// TIA Portal project "Ejercicio3" (V15.1)

(* hardware
DEVICE "S7-1200 station_2"  S7-1200 Station
   slot 0: "Rack_0"  S7-1200 Rack  Rack  V1.0
   slot 1: "PLC_0"  CPU 1215C AC/DC/Rly  6ES7 215-1BG40-0XB0  V4.2
DEVICE "HMI_0"  KTP700 Basic PN
   slot 0: "HMI_0"  KTP700 Basic PN  6AV2 123-2GB03-0AX0  15.1.0.0
   slot 1: "HMI_RT_1"  KTP700 Basic PN  6AV2 123-2GB03-0AX0  15.1.0.0
   slot 5: "HMI_0.IE_CP_1"  PROFINET Interface  15.0.1.0
      slot 1: "Interfaz PROFINET_1"  PROFINET Interface
         slot 1: "Port_1"  Port
*)

// ===== PLC "PLC_0"  CPU 1215C AC/DC/Rly =====

VAR_GLOBAL   // PLC tag table "Tabla de variables estándar"
   "Marcha" AT %M0.0 : Bool;
   "Paro" AT %M0.1 : Bool;
   "Pila de pales en la entrada" AT %M0.2 : Bool;
   "Pila de pale en desapilador" AT %M0.3 : Bool;
   "Palé en rodillos de salida" AT %M0.4 : Bool;
   "Cilindro subir pilas pales reposo" AT %M0.5 : Bool;
   "Cilindro subir pilas pales arriba" AT %M0.6 : Bool;
   "Cilindro uña sujetar pila reposo" AT %M0.7 : Bool;
   "Cilindro uña sujetar pila extendida" AT %M1.0 : Bool;
   "Freno pila recogido" AT %M1.1 : Bool;
   "Freno pila extendido" AT %M1.2 : Bool;
   "Motor rodillos entrada pilas" AT %M10.0 : Bool;
   "Motor rodillos desapilador" AT %M10.1 : Bool;
   "Motor rodillos salida de palé" AT %M10.2 : Bool;
   "Cilindro subir pila" AT %M10.3 : Bool;
   "Cilindro uñas sujetar pila" AT %M10.4 : Bool;
   "Cilindro freno" AT %M10.5 : Bool;
   "Permiso de extraccion de palé" AT %M2.0 : Bool;
END_VAR

// folder: System blocks/Program resources

DATA_BLOCK "IEC_Timer_0_DB"   // DB1
{ S7_Optimized_Access := 'TRUE' }
AUTHOR : Simatic
FAMILY : IEC
NAME : IEC_TMR
VERSION : 1.0
// stored: InstanceOfName IEC_TIMER
"IEC_TIMER"
BEGIN
END_DATA_BLOCK

DATA_BLOCK "IEC_Timer_0_DB_1"   // DB2
{ S7_Optimized_Access := 'TRUE' }
AUTHOR : Simatic
FAMILY : IEC
NAME : IEC_TMR
VERSION : 1.0
// stored: InstanceOfName IEC_TIMER
"IEC_TIMER"
BEGIN
END_DATA_BLOCK

DATA_BLOCK "IEC_Timer_0_DB_2"   // DB3
{ S7_Optimized_Access := 'TRUE' }
AUTHOR : Simatic
FAMILY : IEC
NAME : IEC_TMR
VERSION : 1.0
// stored: InstanceOfName IEC_TIMER
"IEC_TIMER"
BEGIN
END_DATA_BLOCK

// folder: (top level)

ORGANIZATION_BLOCK "Main"   // OB1, LAD, ProgramCycle
TITLE = "Main Program Sweep (Cycle)"
{ S7_Optimized_Access := 'TRUE' }
VERSION : 0.1
   VAR_INPUT
      Initial_Call : Bool;   // Initial call of this OB
      Remanence : Bool;   // =True, if remanent data are available
   END_VAR
BEGIN

REGION Network 1
   // Tenemos  un  pulsador  de  marcha  uno  de  paro  para  el  sistema.  Si  se  pulsa  el  paro  la  secuencia  se detiene continuando en el mismo punto cuando se pulse marcha de nuevo.
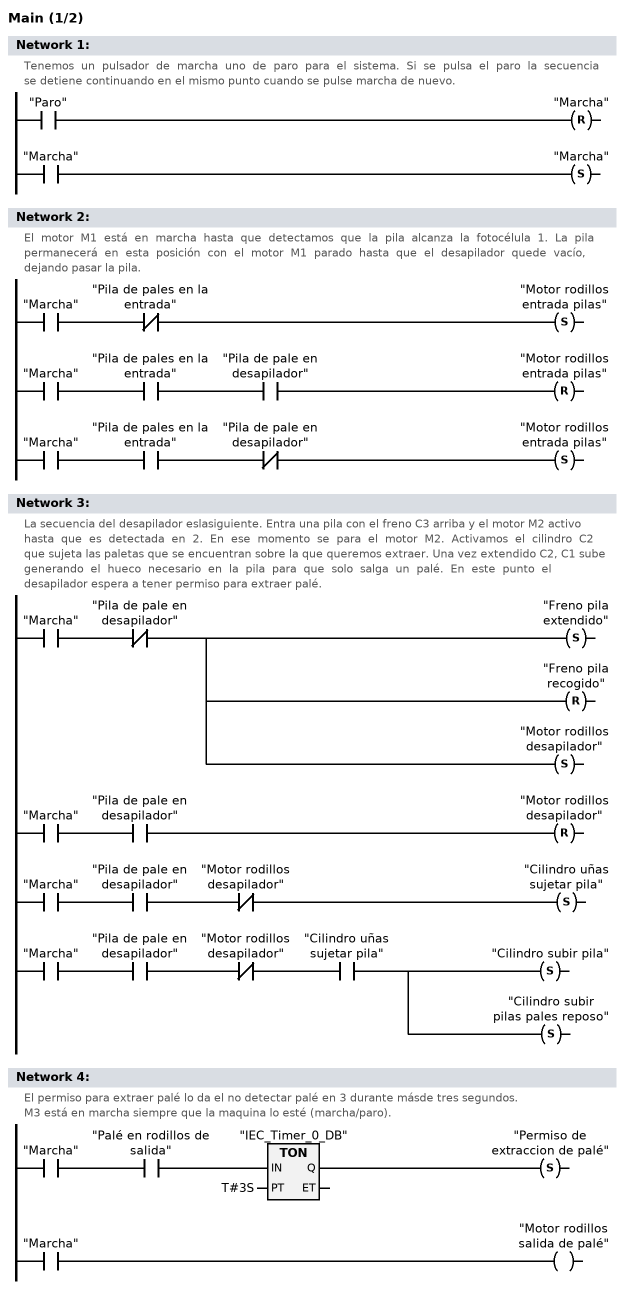
   RUNG wire#powerrail
      Contact( "Paro" )
      R_Coil( "Marcha" )
   END_RUNG
   RUNG wire#powerrail
      Contact( "Marcha" )
      S_Coil( "Marcha" )
   END_RUNG
   // the same network as SCL:
   IF "Paro" THEN "Marcha" := FALSE; END_IF;
   IF "Marcha" THEN "Marcha" := TRUE; END_IF;
END_REGION

REGION Network 2
   // El  motor  M1  está  en  marcha  hasta  que  detectamos  que  la  pila  alcanza  la  fotocélula  1.  La  pila permanecerá  en  esta  posición  con  el  motor  M1  parado  hasta  que  el  desapilador  quede  vacío, dejando pasar la pila.
   RUNG wire#powerrail
      Contact( "Marcha" )
      I_Contact( "Pila de pales en la entrada" )
      S_Coil( "Motor rodillos entrada pilas" )
   END_RUNG
   RUNG wire#powerrail
      Contact( "Marcha" )
      Contact( "Pila de pales en la entrada" )
      Contact( "Pila de pale en desapilador" )
      R_Coil( "Motor rodillos entrada pilas" )
   END_RUNG
   RUNG wire#powerrail
      Contact( "Marcha" )
      Contact( "Pila de pales en la entrada" )
      I_Contact( "Pila de pale en desapilador" )
      S_Coil( "Motor rodillos entrada pilas" )
   END_RUNG
   // the same network as SCL:
   IF "Marcha" AND NOT "Pila de pales en la entrada" THEN "Motor rodillos entrada pilas" := TRUE; END_IF;
   IF "Marcha" AND "Pila de pales en la entrada" AND "Pila de pale en desapilador" THEN
       "Motor rodillos entrada pilas" := FALSE;
   END_IF;
   IF "Marcha" AND "Pila de pales en la entrada" AND NOT "Pila de pale en desapilador" THEN
       "Motor rodillos entrada pilas" := TRUE;
   END_IF;
END_REGION

REGION Network 3
   // La secuencia del desapilador eslasiguiente. Entra una pila con el freno C3 arriba y el motor M2 activo hasta  que  es  detectada  en  2.  En  ese  momento  se  para  el  motor  M2.  Activamos  el  cilindro  C2  que sujeta las paletas que se encuentran sobre la que queremos extraer. Una vez extendido C2, C1 sube generando  el  hueco  necesario  en  la  pila  para  que  solo  salga  un  palé.  En  este  punto  el  desapilador espera a tener permiso para extraer palé.
   RUNG wire#powerrail
      Contact( "Marcha" )
      I_Contact( "Pila de pale en desapilador" )
      wire#w1
      S_Coil( "Freno pila extendido" )
   END_RUNG
   RUNG wire#w1
      R_Coil( "Freno pila recogido" )
   END_RUNG
   RUNG wire#w1
      S_Coil( "Motor rodillos desapilador" )
   END_RUNG
   RUNG wire#powerrail
      Contact( "Marcha" )
      Contact( "Pila de pale en desapilador" )
      R_Coil( "Motor rodillos desapilador" )
   END_RUNG
   RUNG wire#powerrail
      Contact( "Marcha" )
      Contact( "Pila de pale en desapilador" )
      I_Contact( "Motor rodillos desapilador" )
      S_Coil( "Cilindro uñas sujetar pila" )
   END_RUNG
   RUNG wire#powerrail
      Contact( "Marcha" )
      Contact( "Pila de pale en desapilador" )
      I_Contact( "Motor rodillos desapilador" )
      Contact( "Cilindro uñas sujetar pila" )
      wire#w2
      S_Coil( "Cilindro subir pila" )
   END_RUNG
   RUNG wire#w2
      S_Coil( "Cilindro subir pilas pales reposo" )
   END_RUNG
   // the same network as SCL:
   IF "Marcha" AND NOT "Pila de pale en desapilador" THEN
       "Freno pila extendido" := TRUE;
       "Freno pila recogido" := FALSE;
       "Motor rodillos desapilador" := TRUE;
   END_IF;
   IF "Marcha" AND "Pila de pale en desapilador" THEN "Motor rodillos desapilador" := FALSE; END_IF;
   IF "Marcha" AND "Pila de pale en desapilador" AND NOT "Motor rodillos desapilador" THEN
       "Cilindro uñas sujetar pila" := TRUE;
   END_IF;
   IF "Marcha" AND "Pila de pale en desapilador" AND NOT "Motor rodillos desapilador" AND "Cilindro uñas sujetar pila" THEN
       "Cilindro subir pila" := TRUE;
       "Cilindro subir pilas pales reposo" := TRUE;
   END_IF;
END_REGION

REGION Network 4
   // El permiso para extraer palé lo da el no detectar palé en 3 durante másde tres segundos.
   // M3 está en marcha siempre que la maquina lo esté (marcha/paro).
   "IEC_Timer_0_DB".TON(IN := "Marcha" AND "Palé en rodillos de salida", PT := T#3S);
   IF "IEC_Timer_0_DB".Q THEN "Permiso de extraccion de palé" := TRUE; END_IF;
   "Motor rodillos salida de palé" := "Marcha";
END_REGION

REGION Network 5
   // Cuando  el  desapilador  tiene  permiso  para  extraer  el  palé baja  el  freno  C3  activa  el  motor  M2  hasta que  2  no  detecte  paleta  mas  de  3  segundos.  En  ese  momento  entendemos  que  el  palé  ha  salido  y bajamos C1 hastadepositar la pila en el camino de rodillos (4) y entonces desactivamos C2.
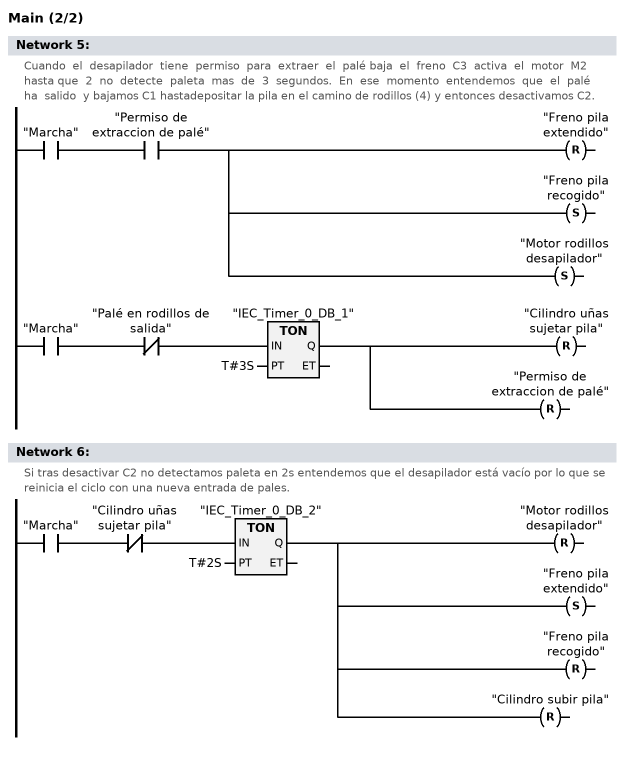
   IF "Marcha" AND "Permiso de extraccion de palé" THEN
       "Freno pila extendido" := FALSE;
       "Freno pila recogido" := TRUE;
       "Motor rodillos desapilador" := TRUE;
   END_IF;
   "IEC_Timer_0_DB_1".TON(IN := "Marcha" AND NOT "Palé en rodillos de salida", PT := T#3S);
   IF "IEC_Timer_0_DB_1".Q THEN
       "Cilindro uñas sujetar pila" := FALSE;
       "Permiso de extraccion de palé" := FALSE;
   END_IF;
END_REGION

REGION Network 6
   // Si tras desactivar C2 no detectamos paleta en 2s entendemos que el desapilador está vacío por lo que se reinicia el ciclo con una nueva entrada de pales.
   "IEC_Timer_0_DB_2".TON(IN := "Marcha" AND NOT "Cilindro uñas sujetar pila", PT := T#2S);
   IF "IEC_Timer_0_DB_2".Q THEN
       "Motor rodillos desapilador" := FALSE;
       "Freno pila extendido" := TRUE;
       "Freno pila recogido" := FALSE;
       "Cilindro subir pila" := FALSE;
   END_IF;
END_REGION
END_ORGANIZATION_BLOCK

(* ===== HMI "HMI_RT_1" =====
system functions are stored by id; their names below are inferred from use
connection "HMI_Conexión_1": ETHERNET, SMART_S7_1200_OMS

HMI tags "Tabla de variables estándar"
   "Número_imagen_variable" : UInt, internal

text list "Nombre_imagen_lista_texto": 1 'Imagen raíz'

Template "Plantilla_1" 800x480
   Button "Salir" at 714,429 size 71x50; TextOff 'Salir'; PictureOff "ExitRuntime_KTP700_Basic_PN_TR"; PictureOn "ExitRuntime_KTP700_Basic_PN_TR"
      on Release: StopRuntime(0)
   Button "Template_Button" at 614,429 size 71x50; TextOff 'Text'
   Button "Template_Button_1" at 514,429 size 71x50; TextOff 'Text'
   Button "Template_Button_2" at 414,429 size 71x50; TextOff 'Text'
   Button "Template_Button_3" at 314,429 size 71x50; TextOff 'Text'
   Button "Template_Button_4" at 214,429 size 71x50; TextOff 'Text'
   Button "Avisos" at 114,429 size 71x50; TextOff 'Avisos'; PictureOff "AlarmDisplay_KTP700_Basic_PN_TR"; PictureOn "AlarmDisplay_KTP700_Basic_PN_TR"
      on Release: function_ef3f5d25("Ventana de avisos_no_acusado", -1)
   Button "Imagen inicial" at 14,429 size 71x50; TextOff 'Imagen inicial'; PictureOff "NavigateHome_KTP700_Basic_PN_TR"; PictureOn "NavigateHome_KTP700_Basic_PN_TR"
      on Release: ActivateScreen("Imagen raíz", 0)
   SymbolicIOField "Imagen_campo_ES_simbólico" at 93,9 size 600x33; TextOff '0'; TextOn '1'; TextList "Nombre_imagen_lista_texto"
      ProcessValue <- "Número_imagen_variable"
      on Change: ActivateScreenByNumber("Número_imagen_variable", 0)
   DateTimeField "HmiScreenItemData" at 695,25 size 105x25
   DateTimeField "HmiScreenItemData_1" at 695,0 size 105x25
   GraphicView "Logotipo" at 0,0 size 91x51; Picture "Logotipo de HMI_1"

screen "Imagen raíz" 800x480, template "Plantilla_1"
   on GenerateScreen: SetTag("Número_imagen_variable", 1)
   Switch "Interruptor_1" at 19,131 size 208x48; CaptionText 'Switch'; TextOff 'OFF'; TextOn 'ON'
   TextField "Campo de texto_1" at 56,82 size 112x39; Text 'Marcha'
   Button "Botón_1" at 16,285 size 211x122; TextOff 'BOTON DE PARO'
   TextField "Campo de texto_2" at 487,93 size 171x28; Text 'Palets en espera'
   TextField "Campo de texto_3" at 487,147 size 221x28; Text 'Palets en desapilador'
   TextField "Campo de texto_4" at 487,207 size 162x28; Text 'Palets en salida'
   TextField "Campo de texto_5" at 492,284 size 132x52; Text 'Estado freno M2 - M3'
   TextField "Campo de texto_6" at 487,353 size 154x52; Text 'Estado cilindro arriba / abajo'
   TextField "Campo de texto_7" at 490,373 size 19x28; Text 'Text'
*)